// TIA Portal V17 export
// export: Created 2024-08-07T21:44:11.3910525Z, ExportSetting WithDefaults, DisplayName Totally Integrated Automation Portal, DisplayVersion V17 Update 7, DisplayName TIA Portal Openness, DisplayVersion V17 Update 7, DisplayName TIA Portal Version Control Interface, DisplayVersion V17, DisplayName SINAMICS Startdrive Advanced, DisplayVersion V17 SP2, DisplayName SINAMICS Startdrive G110M, G120, G120C, G120D, G120P, G115D, DisplayVersion V17 SP2, DisplayName SINAMICS Startdrive G130, G150, S120, S150, SINAMICS MV, S210, DisplayVersion V17 SP2, DisplayName STEP 7 Professional, DisplayVersion V17 Update 7, DisplayName STEP 7 Safety, DisplayVersion V17 Update 6, DisplayName WinCC Advanced / Unified PC, DisplayVersion V17 Update 7
DATA_BLOCK "2. Call_M000_PRODUCTION_DECLARATION_DB"   // DB2003
VERSION : 0.1
// stored: AutoNumber false, DBAccessibleFromOPCUA true, DBAccessibleFromWebserver true, InstanceOfName 2. Call_M000_PRODUCTION_DECLARATION, InstanceOfType FB
"2. Call_M000_PRODUCTION_DECLARATION"
   // VAR_INPUT
   //    CYCLE_COUNTER : DInt;
   // END_VAR
   // VAR_IN_OUT
   //    LOCAL_PART_ARRAY : Variant;
   //    LOCAL_PART_WSTRING : Variant;
   //    LOCAL_TOOL : Variant;
   //    TRACA_REF : Variant;
   //    QUANTITY : Variant;
   //    STATION_NAME : Variant;
   // END_VAR
   // VAR
   //    cycleCounter_temp : DInt;
   //    LOCAL_PART_OK : WString;
   //    STATION_NAME_OK : WString;
   //    aux : Struct
   //       idx : UInt;
   //       cnt : UInt;
   //       sizeCnt : Bool;
   //       LOCAL_PART_STRING : String;
   //    END_STRUCT;
   // END_VAR
BEGIN
END_DATA_BLOCK
